(* Logix 5000 project; controller Timers Emulate 5570 rev 33.11; software revision 33.00 *)

TASK T00_MainTask (continuous, watchdog 500 ms) : P00_MainProgram

MODULES
   Local : Emulate 5570 (ICP 2, rev 33.11)
END_MODULES

PROGRAM P00_MainProgram   (* main routine R00_MainRoutine *)
VAR
   B01_Activacion_Alarma : BOOL;   // Bandera de activacion de Alarma
   ES : BOOL;   // Boton de Paro de emergencia
   I01_Desactivar_Alarma : BOOL;   // Boton para desactivar Alarma
   O01_Lampara : BOOL;   // Luz de seguridad
   O02_Alarma : BOOL;   // Alarma
   O03_P : BOOL;
   S01_Movimiento : BOOL;   // Sensor de Movimiento
   T01_DesactivarLuz : TIMER := (PRE := 10000);   // Timer para desactivar luz en 10s
   T02_Alarma : TIMER := (PRE := 5000);   // Activacion de Alarma
   T03_TOF_LUZ : TIMER := (PRE := 10000);
END_VAR

ROUTINE R00_MainRoutine   (* ladder *)
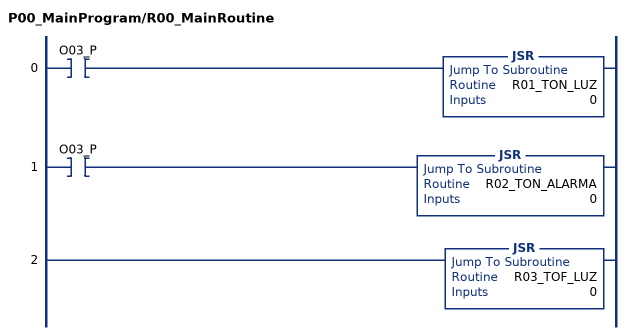
   0: XIC(O03_P)JSR(R01_TON_LUZ,0);
   1: XIC(O03_P)JSR(R02_TON_ALARMA,0);
   2: JSR(R03_TOF_LUZ,0);
END_ROUTINE

ROUTINE R01_TON_LUZ   (* ladder *)
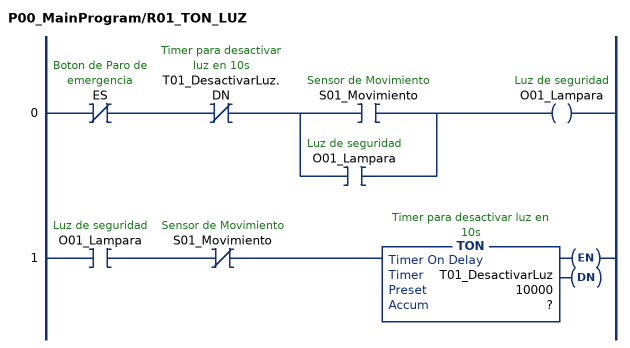
   0: XIO(ES)XIO(T01_DesactivarLuz.DN)[XIC(S01_Movimiento) ,XIC(O01_Lampara) ]OTE(O01_Lampara);
   1: XIC(O01_Lampara)XIO(S01_Movimiento)TON(T01_DesactivarLuz,?,?);
END_ROUTINE

ROUTINE R02_TON_ALARMA   (* ladder *)
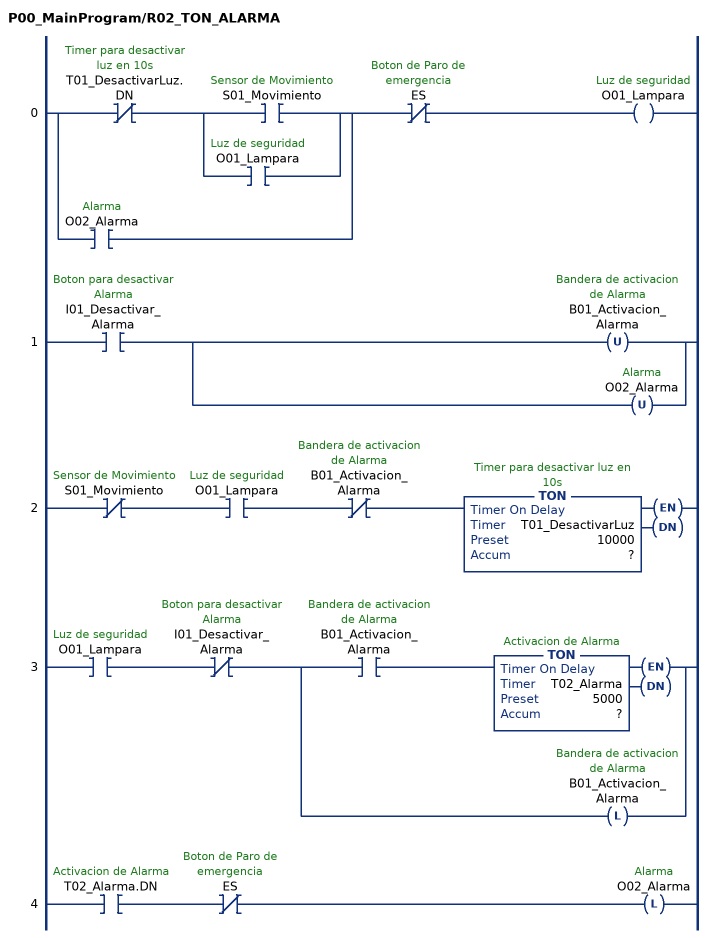
   0: [XIO(T01_DesactivarLuz.DN) [XIC(S01_Movimiento) ,XIC(O01_Lampara) ] ,XIC(O02_Alarma) ]XIO(ES)OTE(O01_Lampara);
   1: XIC(I01_Desactivar_Alarma)[OTU(B01_Activacion_Alarma) ,OTU(O02_Alarma) ];
   2: XIO(S01_Movimiento)XIC(O01_Lampara)XIO(B01_Activacion_Alarma)TON(T01_DesactivarLuz,?,?);
   3: XIC(O01_Lampara)XIO(I01_Desactivar_Alarma)[XIC(B01_Activacion_Alarma) TON(T02_Alarma,?,?) ,OTL(B01_Activacion_Alarma) ];
   4: XIC(T02_Alarma.DN)XIO(ES)OTL(O02_Alarma);
END_ROUTINE

ROUTINE R03_TOF_LUZ   (* ladder *)
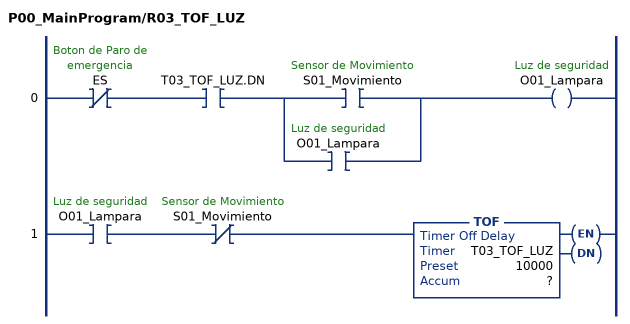
   0: XIO(ES)XIC(T03_TOF_LUZ.DN)[XIC(S01_Movimiento) ,XIC(O01_Lampara) ]OTE(O01_Lampara);
   1: XIC(O01_Lampara)XIO(S01_Movimiento)TOF(T03_TOF_LUZ,?,?);
END_ROUTINE
END_PROGRAM
